{attribute 'qualified_only'}
{attribute 'strict'}
{attribute 'to_string'}
TYPE eMessageCategories :
(
	None:=0,	
	TimeoutFailure := 1,
	MissingData := 2,
	LostConnection := 3,
	Undefined := 4,
	NotImplemented:=5,
	NotAllowed:=6,
	ParentFailed:=7,
	External:=8,
	Positiv:=9,
	StateMachine:=10,
	HardwareFailure := 11,
	ChildFailed := 12
);
END_TYPE

(* stored: Version 1.1.0.1, ProductVersion 3.1.4026.18
   DUT eMessageCategories: Id {f686d474-7d27-4531-ac7a-80c2a5b3adc0} *)
